FUNCTION_BLOCK FB_Word_To_Bool
VAR_INPUT
	inWord : WORD;
END_VAR
VAR_OUTPUT
	outArrayOfBool : ARRAY [0..15] OF BOOL;
END_VAR
VAR
END_VAR

outArrayOfBool[0] := inWord.0;
outArrayOfBool[1] := inWord.1;
outArrayOfBool[2] := inWord.2;
outArrayOfBool[3] := inWord.3;
outArrayOfBool[4] := inWord.4;
outArrayOfBool[5] := inWord.5;
outArrayOfBool[6] := inWord.6;
outArrayOfBool[7] := inWord.7;
outArrayOfBool[8] := inWord.8;
outArrayOfBool[9] := inWord.9;
outArrayOfBool[10] := inWord.10;
outArrayOfBool[11] := inWord.11;
outArrayOfBool[12] := inWord.12;
outArrayOfBool[13] := inWord.13;
outArrayOfBool[14] := inWord.14;
outArrayOfBool[15] := inWord.15;

END_FUNCTION_BLOCK

(* stored: Version 1.1.0.1, ProductVersion 3.1.4024.11
   POU FB_Word_To_Bool: Id {d3d8282c-3aea-460d-99cc-fe2a8ba427ea}, SpecialFunc None *)
